(* IEC 61131-3 sources: repolevel_ST_code_completion/dataset/generation_context_ground_truth/TestMQTTGithubInterfaceExamplePayload, 4 files *)

(* ---- StringReciver.st ---- *)
VAR
	//from this instance i can get my string...
	MQTTString:MQTT.ReceiveString;
	init: BOOL;
	{attribute 'instance-path'}
	{attribute 'noinit'}
	instanceName: STRING(255);//this string contains the instance name of the FB
	//here we get the "lowest" element of the name...
	LastTreeName:STRING;
	StringPointer:POINTER TO STRING;
END_VAR

IF NOT init THEN
	init := TRUE;
	StringPointer := CommonTypesAndFunctions.FindLastDot(ADR(instanceName));

	StringPointer := StringPointer + SIZEOF(BYTE);

	LastTreeName := StringPointer^;
	MQTTString.initAsFindPayload(compString:=ADR(LastTreeName), returnHit:= TRUE, splitChar:= ':');
END_IF

(* ---- StringReciver_PublishReceived.st ---- *)
VAR
	//from this instance i can get my string...
	MQTTString:MQTT.ReceiveString;
	init: BOOL;
	{attribute 'instance-path'}
	{attribute 'noinit'}
	instanceName: STRING(255);//this string contains the instance name of the FB
	//here we get the "lowest" element of the name...
	LastTreeName:STRING;
	StringPointer:POINTER TO STRING;
END_VAR

PublishReceived := MQTTString.PublishReceived(Data:= Data);

(* ---- ValueReciver.st ---- *)
VAR
	//from this instance i can get my value...
	MQTTValue:MQTT.ReceiveValue;
	init: BOOL;
	{attribute 'instance-path'}
	{attribute 'noinit'}
	instanceName: STRING(255);//this string contains the instance name of the FB
	//here we get the "lowest" element of the name...
	LastTreeName:STRING;
	StringPointer:POINTER TO STRING;
END_VAR

IF NOT init THEN
	init := TRUE;
	StringPointer := CommonTypesAndFunctions.FindLastDot(ADR(instanceName));

	StringPointer := StringPointer + SIZEOF(BYTE);

	LastTreeName := StringPointer^;
	MQTTValue.initAsFindPayload(compString:=ADR(LastTreeName), returnHit:= TRUE, ValueTyp:= IBaseLibrary.TYPE_LREAL, splitChar:= ':');
END_IF

(* ---- ValueReciver_PublishReceived.st ---- *)
VAR
	//from this instance i can get my value...
	MQTTValue:MQTT.ReceiveValue;
	init: BOOL;
	{attribute 'instance-path'}
	{attribute 'noinit'}
	instanceName: STRING(255);//this string contains the instance name of the FB
	//here we get the "lowest" element of the name...
	LastTreeName:STRING;
	StringPointer:POINTER TO STRING;
END_VAR

PublishReceived := MQTTValue.PublishReceived(Data:= Data);
